TYPE ScreenConfigs :
STRUCT
	DM430GNScreenConfigFS : DM430GNScreenConfig;
	DM430GNScreenConfigBS : DM430GNScreenConfig;
END_STRUCT
END_TYPE

(* stored: Version 1.1.0.1, ProductVersion 3.1.4024.12
   DUT ScreenConfigs: Id {1cd767aa-8cbd-4ff5-aa47-eac5c7084061} *)
